  583 = 'S3 583 Row 59 Lost Return Position... Check Ixxx.x Default' | German: 'S3 583 Row 59 Lost Return Position... Check Ixxx.x German' | French: 'S3 583 Row 59 Lost Return Position... Check Ixxx.x French'
  584 = 'S3 584 Row 59 Switch Fault... Check Ixxx.x / Ixxx.x Default' | German: 'S3 584 Row 59 Switch Fault... Check Ixxx.x / Ixxx.x German' | French: 'S3 584 Row 59 Switch Fault... Check Ixxx.x / Ixxx.x French'
  585 = 'S3 585 Row 59 Spare Message Default' | German: 'S3 585 Row 59 Spare Message German' | French: 'S3 585 Row 59 Spare Message French'
  586 = 'S3 586 Row 59 Spare Message Default' | German: 'S3 586 Row 59 Spare Message German' | French: 'S3 586 Row 59 Spare Message French'
  587 = 'S3 587 Row 59 Spare Message Default' | German: 'S3 587 Row 59 Spare Message German' | French: 'S3 587 Row 59 Spare Message French'
  588 = 'S3 588 Row 59 Spare Message Default' | German: 'S3 588 Row 59 Spare Message German' | French: 'S3 588 Row 59 Spare Message French'
  589 = 'S3 589 Row 59 Spare Message Default' | German: 'S3 589 Row 59 Spare Message German' | French: 'S3 589 Row 59 Spare Message French'
  590 = 'S3 590 Row 60 Failed To Advance.. Check Qxxx.x Default' | German: 'S3 590 Row 60 Failed To Advance.. Check Qxxx.x German' | French: 'S3 590 Row 60 Failed To Advance.. Check Qxxx.x French'
  591 = 'S3 591 Row 60 Failed To Return.. Check Qxxx.x Default' | German: 'S3 591 Row 60 Failed To Return.. Check Qxxx.x German' | French: 'S3 591 Row 60 Failed To Return.. Check Qxxx.x French'
  592 = 'S3 592 Row 60 Lost Advance Position... Check Ixxx.x Default' | German: 'S3 592 Row 60 Lost Advance Position... Check Ixxx.x German' | French: 'S3 592 Row 60 Lost Advance Position... Check Ixxx.x French'
  593 = 'S3 593 Row 60 Lost Return Position... Check Ixxx.x Default' | German: 'S3 593 Row 60 Lost Return Position... Check Ixxx.x German' | French: 'S3 593 Row 60 Lost Return Position... Check Ixxx.x French'
  594 = 'S3 594 Row 60 Switch Fault... Check Ixxx.x / Ixxx.x Default' | German: 'S3 594 Row 60 Switch Fault... Check Ixxx.x / Ixxx.x German' | French: 'S3 594 Row 60 Switch Fault... Check Ixxx.x / Ixxx.x French'
  595 = 'S3 595 Row 60 Spare Message Default' | German: 'S3 595 Row 60 Spare Message German' | French: 'S3 595 Row 60 Spare Message French'
  596 = 'S3 596 Row 60 Spare Message Default' | German: 'S3 596 Row 60 Spare Message German' | French: 'S3 596 Row 60 Spare Message French'
  597 = 'S3 597 Row 60 Spare Message Default' | German: 'S3 597 Row 60 Spare Message German' | French: 'S3 597 Row 60 Spare Message French'
  598 = 'S3 598 Row 60 Spare Message Default' | German: 'S3 598 Row 60 Spare Message German' | French: 'S3 598 Row 60 Spare Message French'
  599 = 'S3 599 Row 60 Spare Message Default' | German: 'S3 599 Row 60 Spare Message German' | French: 'S3 599 Row 60 Spare Message French'
  600 = 'S3 600 Row 61 Failed To Advance.. Check Qxxx.x Default' | German: 'S3 600 Row 61 Failed To Advance.. Check Qxxx.x German' | French: 'S3 600 Row 61 Failed To Advance.. Check Qxxx.x French'
  601 = 'S3 601 Row 61 Failed To Return.. Check Qxxx.x Default' | German: 'S3 601 Row 61 Failed To Return.. Check Qxxx.x German' | French: 'S3 601 Row 61 Failed To Return.. Check Qxxx.x French'
  602 = 'S3 602 Row 61 Lost Advance Position... Check Ixxx.x Default' | German: 'S3 602 Row 61 Lost Advance Position... Check Ixxx.x German' | French: 'S3 602 Row 61 Lost Advance Position... Check Ixxx.x French'
  603 = 'S3 603 Row 61 Lost Return Position... Check Ixxx.x Default' | German: 'S3 603 Row 61 Lost Return Position... Check Ixxx.x German' | French: 'S3 603 Row 61 Lost Return Position... Check Ixxx.x French'
  604 = 'S3 604 Row 61 Switch Fault... Check Ixxx.x / Ixxx.x Default' | German: 'S3 604 Row 61 Switch Fault... Check Ixxx.x / Ixxx.x German' | French: 'S3 604 Row 61 Switch Fault... Check Ixxx.x / Ixxx.x French'
  605 = 'S3 605 Row 61 Spare Message Default' | German: 'S3 605 Row 61 Spare Message German' | French: 'S3 605 Row 61 Spare Message French'
  606 = 'S3 606 Row 61 Spare Message Default' | German: 'S3 606 Row 61 Spare Message German' | French: 'S3 606 Row 61 Spare Message French'
  607 = 'S3 607 Row 61 Spare Message Default' | German: 'S3 607 Row 61 Spare Message German' | French: 'S3 607 Row 61 Spare Message French'
  608 = 'S3 608 Row 61 Spare Message Default' | German: 'S3 608 Row 61 Spare Message German' | French: 'S3 608 Row 61 Spare Message French'
  609 = 'S3 609 Row 61 Spare Message Default' | German: 'S3 609 Row 61 Spare Message German' | French: 'S3 609 Row 61 Spare Message French'
  610 = 'S3 610 Row 62 Failed To Advance.. Check Qxxx.x Default' | German: 'S3 610 Row 62 Failed To Advance.. Check Qxxx.x German' | French: 'S3 610 Row 62 Failed To Advance.. Check Qxxx.x French'
  611 = 'S3 611 Row 62 Failed To Return.. Check Qxxx.x Default' | German: 'S3 611 Row 62 Failed To Return.. Check Qxxx.x German' | French: 'S3 611 Row 62 Failed To Return.. Check Qxxx.x French'
  612 = 'S3 612 Row 62 Lost Advance Position... Check Ixxx.x Default' | German: 'S3 612 Row 62 Lost Advance Position... Check Ixxx.x German' | French: 'S3 612 Row 62 Lost Advance Position... Check Ixxx.x French'
  613 = 'S3 613 Row 62 Lost Return Position... Check Ixxx.x Default' | German: 'S3 613 Row 62 Lost Return Position... Check Ixxx.x German' | French: 'S3 613 Row 62 Lost Return Position... Check Ixxx.x French'
  614 = 'S3 614 Row 62 Switch Fault... Check Ixxx.x / Ixxx.x Default' | German: 'S3 614 Row 62 Switch Fault... Check Ixxx.x / Ixxx.x German' | French: 'S3 614 Row 62 Switch Fault... Check Ixxx.x / Ixxx.x French'
  615 = 'S3 615 Row 62 Spare Message Default' | German: 'S3 615 Row 62 Spare Message German' | French: 'S3 615 Row 62 Spare Message French'
  616 = 'S3 616 Row 62 Spare Message Default' | German: 'S3 616 Row 62 Spare Message German' | French: 'S3 616 Row 62 Spare Message French'
  617 = 'S3 617 Row 62 Spare Message Default' | German: 'S3 617 Row 62 Spare Message German' | French: 'S3 617 Row 62 Spare Message French'
  618 = 'S3 618 Row 62 Spare Message Default' | German: 'S3 618 Row 62 Spare Message German' | French: 'S3 618 Row 62 Spare Message French'
  619 = 'S3 619 Row 62 Spare Message Default' | German: 'S3 619 Row 62 Spare Message German' | French: 'S3 619 Row 62 Spare Message French'
  620 = 'S3 620 Row 63 Failed To Advance.. Check Qxxx.x Default' | German: 'S3 620 Row 63 Failed To Advance.. Check Qxxx.x German' | French: 'S3 620 Row 63 Failed To Advance.. Check Qxxx.x French'
  621 = 'S3 621 Row 63 Failed To Return.. Check Qxxx.x Default' | German: 'S3 621 Row 63 Failed To Return.. Check Qxxx.x German' | French: 'S3 621 Row 63 Failed To Return.. Check Qxxx.x French'
  622 = 'S3 622 Row 63 Lost Advance Position... Check Ixxx.x Default' | German: 'S3 622 Row 63 Lost Advance Position... Check Ixxx.x German' | French: 'S3 622 Row 63 Lost Advance Position... Check Ixxx.x French'
  623 = 'S3 623 Row 63 Lost Return Position... Check Ixxx.x Default' | German: 'S3 623 Row 63 Lost Return Position... Check Ixxx.x German' | French: 'S3 623 Row 63 Lost Return Position... Check Ixxx.x French'
  624 = 'S3 624 Row 63 Switch Fault... Check Ixxx.x / Ixxx.x Default' | German: 'S3 624 Row 63 Switch Fault... Check Ixxx.x / Ixxx.x German' | French: 'S3 624 Row 63 Switch Fault... Check Ixxx.x / Ixxx.x French'
  625 = 'S3 625 Row 63 Spare Message Default' | German: 'S3 625 Row 63 Spare Message German' | French: 'S3 625 Row 63 Spare Message French'
  626 = 'S3 626 Row 63 Spare Message Default' | German: 'S3 626 Row 63 Spare Message German' | French: 'S3 626 Row 63 Spare Message French'
  627 = 'S3 627 Row 63 Spare Message Default' | German: 'S3 627 Row 63 Spare Message German' | French: 'S3 627 Row 63 Spare Message French'
  628 = 'S3 628 Row 63 Spare Message Default' | German: 'S3 628 Row 63 Spare Message German' | French: 'S3 628 Row 63 Spare Message French'
  629 = 'S3 629 Row 63 Spare Message Default' | German: 'S3 629 Row 63 Spare Message German' | French: 'S3 629 Row 63 Spare Message French'
  630 = 'S3 630 Row 64 Failed To Advance.. Check Qxxx.x Default' | German: 'S3 630 Row 64 Failed To Advance.. Check Qxxx.x German' | French: 'S3 630 Row 64 Failed To Advance.. Check Qxxx.x French'
  631 = 'S3 631 Row 64 Failed To Return.. Check Qxxx.x Default' | German: 'S3 631 Row 64 Failed To Return.. Check Qxxx.x German' | French: 'S3 631 Row 64 Failed To Return.. Check Qxxx.x French'
  632 = 'S3 632 Row 64 Lost Advance Position... Check Ixxx.x Default' | German: 'S3 632 Row 64 Lost Advance Position... Check Ixxx.x German' | French: 'S3 632 Row 64 Lost Advance Position... Check Ixxx.x French'
  633 = 'S3 633 Row 64 Lost Return Position... Check Ixxx.x Default' | German: 'S3 633 Row 64 Lost Return Position... Check Ixxx.x German' | French: 'S3 633 Row 64 Lost Return Position... Check Ixxx.x French'
  634 = 'S3 634 Row 64 Switch Fault... Check Ixxx.x / Ixxx.x Default' | German: 'S3 634 Row 64 Switch Fault... Check Ixxx.x / Ixxx.x German' | French: 'S3 634 Row 64 Switch Fault... Check Ixxx.x / Ixxx.x French'
  635 = 'S3 635 Row 64 Spare Message Default' | German: 'S3 635 Row 64 Spare Message German' | French: 'S3 635 Row 64 Spare Message French'
  636 = 'S3 636 Row 64 Spare Message Default' | German: 'S3 636 Row 64 Spare Message German' | French: 'S3 636 Row 64 Spare Message French'
  637 = 'S3 637 Row 64 Spare Message Default' | German: 'S3 637 Row 64 Spare Message German' | French: 'S3 637 Row 64 Spare Message French'
  638 = 'S3 638 Row 64 Spare Message Default' | German: 'S3 638 Row 64 Spare Message German' | French: 'S3 638 Row 64 Spare Message French'
  639 = 'S3 639 Row 64 Spare Message Default' | German: 'S3 639 Row 64 Spare Message German' | French: 'S3 639 Row 64 Spare Message French'
  640 = 'S3 640 Row 65 Failed To Advance.. Check Qxxx.x Default' | German: 'S3 640 Row 65 Failed To Advance.. Check Qxxx.x German' | French: 'S3 640 Row 65 Failed To Advance.. Check Qxxx.x French'
  641 = 'S3 641 Row 65 Failed To Return.. Check Qxxx.x Default' | German: 'S3 641 Row 65 Failed To Return.. Check Qxxx.x German' | French: 'S3 641 Row 65 Failed To Return.. Check Qxxx.x French'
  642 = 'S3 642 Row 65 Lost Advance Position... Check Ixxx.x Default' | German: 'S3 642 Row 65 Lost Advance Position... Check Ixxx.x German' | French: 'S3 642 Row 65 Lost Advance Position... Check Ixxx.x French'
  643 = 'S3 643 Row 65 Lost Return Position... Check Ixxx.x Default' | German: 'S3 643 Row 65 Lost Return Position... Check Ixxx.x German' | French: 'S3 643 Row 65 Lost Return Position... Check Ixxx.x French'
  644 = 'S3 644 Row 65 Switch Fault... Check Ixxx.x / Ixxx.x Default' | German: 'S3 644 Row 65 Switch Fault... Check Ixxx.x / Ixxx.x German' | French: 'S3 644 Row 65 Switch Fault... Check Ixxx.x / Ixxx.x French'
  645 = 'S3 645 Row 65 Spare Message Default' | German: 'S3 645 Row 65 Spare Message German' | French: 'S3 645 Row 65 Spare Message French'
  646 = 'S3 646 Row 65 Spare Message Default' | German: 'S3 646 Row 65 Spare Message German' | French: 'S3 646 Row 65 Spare Message French'
  647 = 'S3 647 Row 65 Spare Message Default' | German: 'S3 647 Row 65 Spare Message German' | French: 'S3 647 Row 65 Spare Message French'
  648 = 'S3 648 Row 65 Spare Message Default' | German: 'S3 648 Row 65 Spare Message German' | French: 'S3 648 Row 65 Spare Message French'
  649 = 'S3 649 Row 65 Spare Message Default' | German: 'S3 649 Row 65 Spare Message German' | French: 'S3 649 Row 65 Spare Message French'
  650 = 'S3 650 Row 66 Failed To Advance.. Check Qxxx.x Default' | German: 'S3 650 Row 66 Failed To Advance.. Check Qxxx.x German' | French: 'S3 650 Row 66 Failed To Advance.. Check Qxxx.x French'
  651 = 'S3 651 Row 66 Failed To Return.. Check Qxxx.x Default' | German: 'S3 651 Row 66 Failed To Return.. Check Qxxx.x German' | French: 'S3 651 Row 66 Failed To Return.. Check Qxxx.x French'
  652 = 'S3 652 Row 66 Lost Advance Position... Check Ixxx.x Default' | German: 'S3 652 Row 66 Lost Advance Position... Check Ixxx.x German' | French: 'S3 652 Row 66 Lost Advance Position... Check Ixxx.x French'
  653 = 'S3 653 Row 66 Lost Return Position... Check Ixxx.x Default' | German: 'S3 653 Row 66 Lost Return Position... Check Ixxx.x German' | French: 'S3 653 Row 66 Lost Return Position... Check Ixxx.x French'
  654 = 'S3 654 Row 66 Switch Fault... Check Ixxx.x / Ixxx.x Default' | German: 'S3 654 Row 66 Switch Fault... Check Ixxx.x / Ixxx.x German' | French: 'S3 654 Row 66 Switch Fault... Check Ixxx.x / Ixxx.x French'
  655 = 'S3 655 Row 66 Spare Message Default' | German: 'S3 655 Row 66 Spare Message German' | French: 'S3 655 Row 66 Spare Message French'
  656 = 'S3 656 Row 66 Spare Message Default' | German: 'S3 656 Row 66 Spare Message German' | French: 'S3 656 Row 66 Spare Message French'
  657 = 'S3 657 Row 66 Spare Message Default' | German: 'S3 657 Row 66 Spare Message German' | French: 'S3 657 Row 66 Spare Message French'
  658 = 'S3 658 Row 66 Spare Message Default' | German: 'S3 658 Row 66 Spare Message German' | French: 'S3 658 Row 66 Spare Message French'
  659 = 'S3 659 Row 66 Spare Message Default' | German: 'S3 659 Row 66 Spare Message German' | French: 'S3 659 Row 66 Spare Message French'
  660 = 'S3 660 Row 67 Failed To Advance.. Check Qxxx.x Default' | German: 'S3 660 Row 67 Failed To Advance.. Check Qxxx.x German' | French: 'S3 660 Row 67 Failed To Advance.. Check Qxxx.x French'
  661 = 'S3 661 Row 67 Failed To Return.. Check Qxxx.x Default' | German: 'S3 661 Row 67 Failed To Return.. Check Qxxx.x German' | French: 'S3 661 Row 67 Failed To Return.. Check Qxxx.x French'
  662 = 'S3 662 Row 67 Lost Advance Position... Check Ixxx.x Default' | German: 'S3 662 Row 67 Lost Advance Position... Check Ixxx.x German' | French: 'S3 662 Row 67 Lost Advance Position... Check Ixxx.x French'
  663 = 'S3 663 Row 67 Lost Return Position... Check Ixxx.x Default' | German: 'S3 663 Row 67 Lost Return Position... Check Ixxx.x German' | French: 'S3 663 Row 67 Lost Return Position... Check Ixxx.x French'
  664 = 'S3 664 Row 67 Switch Fault... Check Ixxx.x / Ixxx.x Default' | German: 'S3 664 Row 67 Switch Fault... Check Ixxx.x / Ixxx.x German' | French: 'S3 664 Row 67 Switch Fault... Check Ixxx.x / Ixxx.x French'
  665 = 'S3 665 Row 67 Spare Message Default' | German: 'S3 665 Row 67 Spare Message German' | French: 'S3 665 Row 67 Spare Message French'
  666 = 'S3 666 Row 67 Spare Message Default' | German: 'S3 666 Row 67 Spare Message German' | French: 'S3 666 Row 67 Spare Message French'
  667 = 'S3 667 Row 67 Spare Message Default' | German: 'S3 667 Row 67 Spare Message German' | French: 'S3 667 Row 67 Spare Message French'
  668 = 'S3 668 Row 67 Spare Message Default' | German: 'S3 668 Row 67 Spare Message German' | French: 'S3 668 Row 67 Spare Message French'
  669 = 'S3 669 Row 67 Spare Message Default' | German: 'S3 669 Row 67 Spare Message German' | French: 'S3 669 Row 67 Spare Message French'
  670 = 'S3 670 Row 68 Failed To Advance.. Check Qxxx.x Default' | German: 'S3 670 Row 68 Failed To Advance.. Check Qxxx.x German' | French: 'S3 670 Row 68 Failed To Advance.. Check Qxxx.x French'
  671 = 'S3 671 Row 68 Failed To Return.. Check Qxxx.x Default' | German: 'S3 671 Row 68 Failed To Return.. Check Qxxx.x German' | French: 'S3 671 Row 68 Failed To Return.. Check Qxxx.x French'
  672 = 'S3 672 Row 68 Lost Advance Position... Check Ixxx.x Default' | German: 'S3 672 Row 68 Lost Advance Position... Check Ixxx.x German' | French: 'S3 672 Row 68 Lost Advance Position... Check Ixxx.x French'
  673 = 'S3 673 Row 68 Lost Return Position... Check Ixxx.x Default' | German: 'S3 673 Row 68 Lost Return Position... Check Ixxx.x German' | French: 'S3 673 Row 68 Lost Return Position... Check Ixxx.x French'
  674 = 'S3 674 Row 68 Switch Fault... Check Ixxx.x / Ixxx.x Default' | German: 'S3 674 Row 68 Switch Fault... Check Ixxx.x / Ixxx.x German' | French: 'S3 674 Row 68 Switch Fault... Check Ixxx.x / Ixxx.x French'
  675 = 'S3 675 Row 68 Spare Message Default' | German: 'S3 675 Row 68 Spare Message German' | French: 'S3 675 Row 68 Spare Message French'
  676 = 'S3 676 Row 68 Spare Message Default' | German: 'S3 676 Row 68 Spare Message German' | French: 'S3 676 Row 68 Spare Message French'
  677 = 'S3 677 Row 68 Spare Message Default' | German: 'S3 677 Row 68 Spare Message German' | French: 'S3 677 Row 68 Spare Message French'
  678 = 'S3 678 Row 68 Spare Message Default' | German: 'S3 678 Row 68 Spare Message German' | French: 'S3 678 Row 68 Spare Message French'
  679 = 'S3 679 Row 68 Spare Message Default' | German: 'S3 679 Row 68 Spare Message German' | French: 'S3 679 Row 68 Spare Message French'
  680 = 'S3 680 Row 69 Failed To Advance.. Check Qxxx.x Default' | German: 'S3 680 Row 69 Failed To Advance.. Check Qxxx.x German' | French: 'S3 680 Row 69 Failed To Advance.. Check Qxxx.x French'
  681 = 'S3 681 Row 69 Failed To Return.. Check Qxxx.x Default' | German: 'S3 681 Row 69 Failed To Return.. Check Qxxx.x German' | French: 'S3 681 Row 69 Failed To Return.. Check Qxxx.x French'
  682 = 'S3 682 Row 69 Lost Advance Position... Check Ixxx.x Default' | German: 'S3 682 Row 69 Lost Advance Position... Check Ixxx.x German' | French: 'S3 682 Row 69 Lost Advance Position... Check Ixxx.x French'
  683 = 'S3 683 Row 69 Lost Return Position... Check Ixxx.x Default' | German: 'S3 683 Row 69 Lost Return Position... Check Ixxx.x German' | French: 'S3 683 Row 69 Lost Return Position... Check Ixxx.x French'
  684 = 'S3 684 Row 69 Switch Fault... Check Ixxx.x / Ixxx.x Default' | German: 'S3 684 Row 69 Switch Fault... Check Ixxx.x / Ixxx.x German' | French: 'S3 684 Row 69 Switch Fault... Check Ixxx.x / Ixxx.x French'
  685 = 'S3 685 Row 69 Spare Message Default' | German: 'S3 685 Row 69 Spare Message German' | French: 'S3 685 Row 69 Spare Message French'
  686 = 'S3 686 Row 69 Spare Message Default' | German: 'S3 686 Row 69 Spare Message German' | French: 'S3 686 Row 69 Spare Message French'
  687 = 'S3 687 Row 69 Spare Message Default' | German: 'S3 687 Row 69 Spare Message German' | French: 'S3 687 Row 69 Spare Message French'
  688 = 'S3 688 Row 69 Spare Message Default' | German: 'S3 688 Row 69 Spare Message German' | French: 'S3 688 Row 69 Spare Message French'
  689 = 'S3 689 Row 69 Spare Message Default' | German: 'S3 689 Row 69 Spare Message German' | French: 'S3 689 Row 69 Spare Message French'
  690 = 'S3 690 Row 70 Failed To Advance.. Check Qxxx.x Default' | German: 'S3 690 Row 70 Failed To Advance.. Check Qxxx.x German' | French: 'S3 690 Row 70 Failed To Advance.. Check Qxxx.x French'
  691 = 'S3 691 Row 70 Failed To Return.. Check Qxxx.x Default' | German: 'S3 691 Row 70 Failed To Return.. Check Qxxx.x German' | French: 'S3 691 Row 70 Failed To Return.. Check Qxxx.x French'
  692 = 'S3 692 Row 70 Lost Advance Position... Check Ixxx.x Default' | German: 'S3 692 Row 70 Lost Advance Position... Check Ixxx.x German' | French: 'S3 692 Row 70 Lost Advance Position... Check Ixxx.x French'
  693 = 'S3 693 Row 70 Lost Return Position... Check Ixxx.x Default' | German: 'S3 693 Row 70 Lost Return Position... Check Ixxx.x German' | French: 'S3 693 Row 70 Lost Return Position... Check Ixxx.x French'
  694 = 'S3 694 Row 70 Switch Fault... Check Ixxx.x / Ixxx.x Default' | German: 'S3 694 Row 70 Switch Fault... Check Ixxx.x / Ixxx.x German' | French: 'S3 694 Row 70 Switch Fault... Check Ixxx.x / Ixxx.x French'
  695 = 'S3 695 Row 70 Spare Message Default' | German: 'S3 695 Row 70 Spare Message German' | French: 'S3 695 Row 70 Spare Message French'
  696 = 'S3 696 Row 70 Spare Message Default' | German: 'S3 696 Row 70 Spare Message German' | French: 'S3 696 Row 70 Spare Message French'
  697 = 'S3 697 Row 70 Spare Message Default' | German: 'S3 697 Row 70 Spare Message German' | French: 'S3 697 Row 70 Spare Message French'
  698 = 'S3 698 Row 70 Spare Message Default' | German: 'S3 698 Row 70 Spare Message German' | French: 'S3 698 Row 70 Spare Message French'
  699 = 'S3 699 Row 70 Spare Message Default' | German: 'S3 699 Row 70 Spare Message German' | French: 'S3 699 Row 70 Spare Message French'
  700 = 'S3 700 Row 71 Failed To Advance.. Check Qxxx.x Default' | German: 'S3 700 Row 71 Failed To Advance.. Check Qxxx.x German' | French: 'S3 700 Row 71 Failed To Advance.. Check Qxxx.x French'
  701 = 'S3 701 Row 71 Failed To Return.. Check Qxxx.x Default' | German: 'S3 701 Row 71 Failed To Return.. Check Qxxx.x German' | French: 'S3 701 Row 71 Failed To Return.. Check Qxxx.x French'
  702 = 'S3 702 Row 71 Lost Advance Position... Check Ixxx.x Default' | German: 'S3 702 Row 71 Lost Advance Position... Check Ixxx.x German' | French: 'S3 702 Row 71 Lost Advance Position... Check Ixxx.x French'
  703 = 'S3 703 Row 71 Lost Return Position... Check Ixxx.x Default' | German: 'S3 703 Row 71 Lost Return Position... Check Ixxx.x German' | French: 'S3 703 Row 71 Lost Return Position... Check Ixxx.x French'
  704 = 'S3 704 Row 71 Switch Fault... Check Ixxx.x / Ixxx.x Default' | German: 'S3 704 Row 71 Switch Fault... Check Ixxx.x / Ixxx.x German' | French: 'S3 704 Row 71 Switch Fault... Check Ixxx.x / Ixxx.x French'
  705 = 'S3 705 Row 71 Spare Message Default' | German: 'S3 705 Row 71 Spare Message German' | French: 'S3 705 Row 71 Spare Message French'
  706 = 'S3 706 Row 71 Spare Message Default' | German: 'S3 706 Row 71 Spare Message German' | French: 'S3 706 Row 71 Spare Message French'
  707 = 'S3 707 Row 71 Spare Message Default' | German: 'S3 707 Row 71 Spare Message German' | French: 'S3 707 Row 71 Spare Message French'
  708 = 'S3 708 Row 71 Spare Message Default' | German: 'S3 708 Row 71 Spare Message German' | French: 'S3 708 Row 71 Spare Message French'
  709 = 'S3 709 Row 71 Spare Message Default' | German: 'S3 709 Row 71 Spare Message German' | French: 'S3 709 Row 71 Spare Message French'
  710 = 'S3 710 Row 72 Failed To Advance.. Check Qxxx.x Default' | German: 'S3 710 Row 72 Failed To Advance.. Check Qxxx.x German' | French: 'S3 710 Row 72 Failed To Advance.. Check Qxxx.x French'
  711 = 'S3 711 Row 72 Failed To Return.. Check Qxxx.x Default' | German: 'S3 711 Row 72 Failed To Return.. Check Qxxx.x German' | French: 'S3 711 Row 72 Failed To Return.. Check Qxxx.x French'
  712 = 'S3 712 Row 72 Lost Advance Position... Check Ixxx.x Default' | German: 'S3 712 Row 72 Lost Advance Position... Check Ixxx.x German' | French: 'S3 712 Row 72 Lost Advance Position... Check Ixxx.x French'
  713 = 'S3 713 Row 72 Lost Return Position... Check Ixxx.x Default' | German: 'S3 713 Row 72 Lost Return Position... Check Ixxx.x German' | French: 'S3 713 Row 72 Lost Return Position... Check Ixxx.x French'
  714 = 'S3 714 Row 72 Switch Fault... Check Ixxx.x / Ixxx.x Default' | German: 'S3 714 Row 72 Switch Fault... Check Ixxx.x / Ixxx.x German' | French: 'S3 714 Row 72 Switch Fault... Check Ixxx.x / Ixxx.x French'
  715 = 'S3 715 Row 72 Spare Message Default' | German: 'S3 715 Row 72 Spare Message German' | French: 'S3 715 Row 72 Spare Message French'
  716 = 'S3 716 Row 72 Spare Message Default' | German: 'S3 716 Row 72 Spare Message German' | French: 'S3 716 Row 72 Spare Message French'
  717 = 'S3 717 Row 72 Spare Message Default' | German: 'S3 717 Row 72 Spare Message German' | French: 'S3 717 Row 72 Spare Message French'
  718 = 'S3 718 Row 72 Spare Message Default' | German: 'S3 718 Row 72 Spare Message German' | French: 'S3 718 Row 72 Spare Message French'
  719 = 'S3 719 Row 72 Spare Message Default' | German: 'S3 719 Row 72 Spare Message German' | French: 'S3 719 Row 72 Spare Message French'
  720 = 'S3 720 Row 73 Failed To Advance.. Check Qxxx.x Default' | German: 'S3 720 Row 73 Failed To Advance.. Check Qxxx.x German' | French: 'S3 720 Row 73 Failed To Advance.. Check Qxxx.x French'
  721 = 'S3 721 Row 73 Failed To Return.. Check Qxxx.x Default' | German: 'S3 721 Row 73 Failed To Return.. Check Qxxx.x German' | French: 'S3 721 Row 73 Failed To Return.. Check Qxxx.x French'
  722 = 'S3 722 Row 73 Lost Advance Position... Check Ixxx.x Default' | German: 'S3 722 Row 73 Lost Advance Position... Check Ixxx.x German' | French: 'S3 722 Row 73 Lost Advance Position... Check Ixxx.x French'
  723 = 'S3 723 Row 73 Lost Return Position... Check Ixxx.x Default' | German: 'S3 723 Row 73 Lost Return Position... Check Ixxx.x German' | French: 'S3 723 Row 73 Lost Return Position... Check Ixxx.x French'
  724 = 'S3 724 Row 73 Switch Fault... Check Ixxx.x / Ixxx.x Default' | German: 'S3 724 Row 73 Switch Fault... Check Ixxx.x / Ixxx.x German' | French: 'S3 724 Row 73 Switch Fault... Check Ixxx.x / Ixxx.x French'
  725 = 'S3 725 Row 73 Spare Message Default' | German: 'S3 725 Row 73 Spare Message German' | French: 'S3 725 Row 73 Spare Message French'
  726 = 'S3 726 Row 73 Spare Message Default' | German: 'S3 726 Row 73 Spare Message German' | French: 'S3 726 Row 73 Spare Message French'
  727 = 'S3 727 Row 73 Spare Message Default' | German: 'S3 727 Row 73 Spare Message German' | French: 'S3 727 Row 73 Spare Message French'
  728 = 'S3 728 Row 73 Spare Message Default' | German: 'S3 728 Row 73 Spare Message German' | French: 'S3 728 Row 73 Spare Message French'
  729 = 'S3 729 Row 73 Spare Message Default' | German: 'S3 729 Row 73 Spare Message German' | French: 'S3 729 Row 73 Spare Message French'
  730 = 'S3 730 Row 74 Failed To Advance.. Check Qxxx.x Default' | German: 'S3 730 Row 74 Failed To Advance.. Check Qxxx.x German' | French: 'S3 730 Row 74 Failed To Advance.. Check Qxxx.x French'
  731 = 'S3 731 Row 74 Failed To Return.. Check Qxxx.x Default' | German: 'S3 731 Row 74 Failed To Return.. Check Qxxx.x German' | French: 'S3 731 Row 74 Failed To Return.. Check Qxxx.x French'
  732 = 'S3 732 Row 74 Lost Advance Position... Check Ixxx.x Default' | German: 'S3 732 Row 74 Lost Advance Position... Check Ixxx.x German' | French: 'S3 732 Row 74 Lost Advance Position... Check Ixxx.x French'
  733 = 'S3 733 Row 74 Lost Return Position... Check Ixxx.x Default' | German: 'S3 733 Row 74 Lost Return Position... Check Ixxx.x German' | French: 'S3 733 Row 74 Lost Return Position... Check Ixxx.x French'
  734 = 'S3 734 Row 74 Switch Fault... Check Ixxx.x / Ixxx.x Default' | German: 'S3 734 Row 74 Switch Fault... Check Ixxx.x / Ixxx.x German' | French: 'S3 734 Row 74 Switch Fault... Check Ixxx.x / Ixxx.x French'
  735 = 'S3 735 Row 74 Spare Message Default' | German: 'S3 735 Row 74 Spare Message German' | French: 'S3 735 Row 74 Spare Message French'
  736 = 'S3 736 Row 74 Spare Message Default' | German: 'S3 736 Row 74 Spare Message German' | French: 'S3 736 Row 74 Spare Message French'
  737 = 'S3 737 Row 74 Spare Message Default' | German: 'S3 737 Row 74 Spare Message German' | French: 'S3 737 Row 74 Spare Message French'
  738 = 'S3 738 Row 74 Spare Message Default' | German: 'S3 738 Row 74 Spare Message German' | French: 'S3 738 Row 74 Spare Message French'
  739 = 'S3 739 Row 74 Spare Message Default' | German: 'S3 739 Row 74 Spare Message German' | French: 'S3 739 Row 74 Spare Message French'
  740 = 'S3 740 Row 75 Failed To Advance.. Check Qxxx.x Default' | German: 'S3 740 Row 75 Failed To Advance.. Check Qxxx.x German' | French: 'S3 740 Row 75 Failed To Advance.. Check Qxxx.x French'
  741 = 'S3 741 Row 75 Failed To Return.. Check Qxxx.x Default' | German: 'S3 741 Row 75 Failed To Return.. Check Qxxx.x German' | French: 'S3 741 Row 75 Failed To Return.. Check Qxxx.x French'
  742 = 'S3 742 Row 75 Lost Advance Position... Check Ixxx.x Default' | German: 'S3 742 Row 75 Lost Advance Position... Check Ixxx.x German' | French: 'S3 742 Row 75 Lost Advance Position... Check Ixxx.x French'
  743 = 'S3 743 Row 75 Lost Return Position... Check Ixxx.x Default' | German: 'S3 743 Row 75 Lost Return Position... Check Ixxx.x German' | French: 'S3 743 Row 75 Lost Return Position... Check Ixxx.x French'
  744 = 'S3 744 Row 75 Switch Fault... Check Ixxx.x / Ixxx.x Default' | German: 'S3 744 Row 75 Switch Fault... Check Ixxx.x / Ixxx.x German' | French: 'S3 744 Row 75 Switch Fault... Check Ixxx.x / Ixxx.x French'
  745 = 'S3 745 Row 75 Spare Message Default' | German: 'S3 745 Row 75 Spare Message German' | French: 'S3 745 Row 75 Spare Message French'
  746 = 'S3 746 Row 75 Spare Message Default' | German: 'S3 746 Row 75 Spare Message German' | French: 'S3 746 Row 75 Spare Message French'
  747 = 'S3 747 Row 75 Spare Message Default' | German: 'S3 747 Row 75 Spare Message German' | French: 'S3 747 Row 75 Spare Message French'
  748 = 'S3 748 Row 75 Spare Message Default' | German: 'S3 748 Row 75 Spare Message German' | French: 'S3 748 Row 75 Spare Message French'
  749 = 'S3 749 Row 75 Spare Message Default' | German: 'S3 749 Row 75 Spare Message German' | French: 'S3 749 Row 75 Spare Message French'
  750 = 'S3 750 Row 76 Failed To Advance.. Check Qxxx.x Default' | German: 'S3 750 Row 76 Failed To Advance.. Check Qxxx.x German' | French: 'S3 750 Row 76 Failed To Advance.. Check Qxxx.x French'
  751 = 'S3 751 Row 76 Failed To Return.. Check Qxxx.x Default' | German: 'S3 751 Row 76 Failed To Return.. Check Qxxx.x German' | French: 'S3 751 Row 76 Failed To Return.. Check Qxxx.x French'
  752 = 'S3 752 Row 76 Lost Advance Position... Check Ixxx.x Default' | German: 'S3 752 Row 76 Lost Advance Position... Check Ixxx.x German' | French: 'S3 752 Row 76 Lost Advance Position... Check Ixxx.x French'
  753 = 'S3 753 Row 76 Lost Return Position... Check Ixxx.x Default' | German: 'S3 753 Row 76 Lost Return Position... Check Ixxx.x German' | French: 'S3 753 Row 76 Lost Return Position... Check Ixxx.x French'
  754 = 'S3 754 Row 76 Switch Fault... Check Ixxx.x / Ixxx.x Default' | German: 'S3 754 Row 76 Switch Fault... Check Ixxx.x / Ixxx.x German' | French: 'S3 754 Row 76 Switch Fault... Check Ixxx.x / Ixxx.x French'
  755 = 'S3 755 Row 76 Spare Message Default' | German: 'S3 755 Row 76 Spare Message German' | French: 'S3 755 Row 76 Spare Message French'
  756 = 'S3 756 Row 76 Spare Message Default' | German: 'S3 756 Row 76 Spare Message German' | French: 'S3 756 Row 76 Spare Message French'
  757 = 'S3 757 Row 76 Spare Message Default' | German: 'S3 757 Row 76 Spare Message German' | French: 'S3 757 Row 76 Spare Message French'
  758 = 'S3 758 Row 76 Spare Message Default' | German: 'S3 758 Row 76 Spare Message German' | French: 'S3 758 Row 76 Spare Message French'
  759 = 'S3 759 Row 76 Spare Message Default' | German: 'S3 759 Row 76 Spare Message German' | French: 'S3 759 Row 76 Spare Message French'
  760 = 'S3 760 Row 77 Failed To Advance.. Check Qxxx.x Default' | German: 'S3 760 Row 77 Failed To Advance.. Check Qxxx.x German' | French: 'S3 760 Row 77 Failed To Advance.. Check Qxxx.x French'
  761 = 'S3 761 Row 77 Failed To Return.. Check Qxxx.x Default' | German: 'S3 761 Row 77 Failed To Return.. Check Qxxx.x German' | French: 'S3 761 Row 77 Failed To Return.. Check Qxxx.x French'
  762 = 'S3 762 Row 77 Lost Advance Position... Check Ixxx.x Default' | German: 'S3 762 Row 77 Lost Advance Position... Check Ixxx.x German' | French: 'S3 762 Row 77 Lost Advance Position... Check Ixxx.x French'
  763 = 'S3 763 Row 77 Lost Return Position... Check Ixxx.x Default' | German: 'S3 763 Row 77 Lost Return Position... Check Ixxx.x German' | French: 'S3 763 Row 77 Lost Return Position... Check Ixxx.x French'
  764 = 'S3 764 Row 77 Switch Fault... Check Ixxx.x / Ixxx.x Default' | German: 'S3 764 Row 77 Switch Fault... Check Ixxx.x / Ixxx.x German' | French: 'S3 764 Row 77 Switch Fault... Check Ixxx.x / Ixxx.x French'
  765 = 'S3 765 Row 77 Spare Message Default' | German: 'S3 765 Row 77 Spare Message German' | French: 'S3 765 Row 77 Spare Message French'
  766 = 'S3 766 Row 77 Spare Message Default' | German: 'S3 766 Row 77 Spare Message German' | French: 'S3 766 Row 77 Spare Message French'
  767 = 'S3 767 Row 77 Spare Message Default' | German: 'S3 767 Row 77 Spare Message German' | French: 'S3 767 Row 77 Spare Message French'
  768 = 'S3 768 Row 77 Spare Message Default' | German: 'S3 768 Row 77 Spare Message German' | French: 'S3 768 Row 77 Spare Message French'
  769 = 'S3 769 Row 77 Spare Message Default' | German: 'S3 769 Row 77 Spare Message German' | French: 'S3 769 Row 77 Spare Message French'
  770 = 'S3 770 Row 78 Failed To Advance.. Check Qxxx.x Default' | German: 'S3 770 Row 78 Failed To Advance.. Check Qxxx.x German' | French: 'S3 770 Row 78 Failed To Advance.. Check Qxxx.x French'
  771 = 'S3 771 Row 78 Failed To Return.. Check Qxxx.x Default' | German: 'S3 771 Row 78 Failed To Return.. Check Qxxx.x German' | French: 'S3 771 Row 78 Failed To Return.. Check Qxxx.x French'
  772 = 'S3 772 Row 78 Lost Advance Position... Check Ixxx.x Default' | German: 'S3 772 Row 78 Lost Advance Position... Check Ixxx.x German' | French: 'S3 772 Row 78 Lost Advance Position... Check Ixxx.x French'
  773 = 'S3 773 Row 78 Lost Return Position... Check Ixxx.x Default' | German: 'S3 773 Row 78 Lost Return Position... Check Ixxx.x German' | French: 'S3 773 Row 78 Lost Return Position... Check Ixxx.x French'
  774 = 'S3 774 Row 78 Switch Fault... Check Ixxx.x / Ixxx.x Default' | German: 'S3 774 Row 78 Switch Fault... Check Ixxx.x / Ixxx.x German' | French: 'S3 774 Row 78 Switch Fault... Check Ixxx.x / Ixxx.x French'
  775 = 'S3 775 Row 78 Spare Message Default' | German: 'S3 775 Row 78 Spare Message German' | French: 'S3 775 Row 78 Spare Message French'
  776 = 'S3 776 Row 78 Spare Message Default' | German: 'S3 776 Row 78 Spare Message German' | French: 'S3 776 Row 78 Spare Message French'
  777 = 'S3 777 Row 78 Spare Message Default' | German: 'S3 777 Row 78 Spare Message German' | French: 'S3 777 Row 78 Spare Message French'
  778 = 'S3 778 Row 78 Spare Message Default' | German: 'S3 778 Row 78 Spare Message German' | French: 'S3 778 Row 78 Spare Message French'
  779 = 'S3 779 Row 78 Spare Message Default' | German: 'S3 779 Row 78 Spare Message German' | French: 'S3 779 Row 78 Spare Message French'
  780 = 'S3 780 Row 79 Failed To Advance.. Check Qxxx.x Default' | German: 'S3 780 Row 79 Failed To Advance.. Check Qxxx.x German' | French: 'S3 780 Row 79 Failed To Advance.. Check Qxxx.x French'
  781 = 'S3 781 Row 79 Failed To Return.. Check Qxxx.x Default' | German: 'S3 781 Row 79 Failed To Return.. Check Qxxx.x German' | French: 'S3 781 Row 79 Failed To Return.. Check Qxxx.x French'
  782 = 'S3 782 Row 79 Lost Advance Position... Check Ixxx.x Default' | German: 'S3 782 Row 79 Lost Advance Position... Check Ixxx.x German' | French: 'S3 782 Row 79 Lost Advance Position... Check Ixxx.x French'
  783 = 'S3 783 Row 79 Lost Return Position... Check Ixxx.x Default' | German: 'S3 783 Row 79 Lost Return Position... Check Ixxx.x German' | French: 'S3 783 Row 79 Lost Return Position... Check Ixxx.x French'
  784 = 'S3 784 Row 79 Switch Fault... Check Ixxx.x / Ixxx.x Default' | German: 'S3 784 Row 79 Switch Fault... Check Ixxx.x / Ixxx.x German' | French: 'S3 784 Row 79 Switch Fault... Check Ixxx.x / Ixxx.x French'
  785 = 'S3 785 Row 79 Spare Message Default' | German: 'S3 785 Row 79 Spare Message German' | French: 'S3 785 Row 79 Spare Message French'
  786 = 'S3 786 Row 79 Spare Message Default' | German: 'S3 786 Row 79 Spare Message German' | French: 'S3 786 Row 79 Spare Message French'
  787 = 'S3 787 Row 79 Spare Message Default' | German: 'S3 787 Row 79 Spare Message German' | French: 'S3 787 Row 79 Spare Message French'
  788 = 'S3 788 Row 79 Spare Message Default' | German: 'S3 788 Row 79 Spare Message German' | French: 'S3 788 Row 79 Spare Message French'
  789 = 'S3 789 Row 79 Spare Message Default' | German: 'S3 789 Row 79 Spare Message German' | French: 'S3 789 Row 79 Spare Message French'
  790 = 'S3 790 Row 80 Failed To Advance.. Check Qxxx.x Default' | German: 'S3 790 Row 80 Failed To Advance.. Check Qxxx.x German' | French: 'S3 790 Row 80 Failed To Advance.. Check Qxxx.x French'
  791 = 'S3 791 Row 80 Failed To Return.. Check Qxxx.x Default' | German: 'S3 791 Row 80 Failed To Return.. Check Qxxx.x German' | French: 'S3 791 Row 80 Failed To Return.. Check Qxxx.x French'
  792 = 'S3 792 Row 80 Lost Advance Position... Check Ixxx.x Default' | German: 'S3 792 Row 80 Lost Advance Position... Check Ixxx.x German' | French: 'S3 792 Row 80 Lost Advance Position... Check Ixxx.x French'
  793 = 'S3 793 Row 80 Lost Return Position... Check Ixxx.x Default' | German: 'S3 793 Row 80 Lost Return Position... Check Ixxx.x German' | French: 'S3 793 Row 80 Lost Return Position... Check Ixxx.x French'
  794 = 'S3 794 Row 80 Switch Fault... Check Ixxx.x / Ixxx.x Default' | German: 'S3 794 Row 80 Switch Fault... Check Ixxx.x / Ixxx.x German' | French: 'S3 794 Row 80 Switch Fault... Check Ixxx.x / Ixxx.x French'
  795 = 'S3 795 Row 80 Spare Message Default' | German: 'S3 795 Row 80 Spare Message German' | French: 'S3 795 Row 80 Spare Message French'
  796 = 'S3 796 Row 80 Spare Message Default' | German: 'S3 796 Row 80 Spare Message German' | French: 'S3 796 Row 80 Spare Message French'
  797 = 'S3 797 Row 80 Spare Message Default' | German: 'S3 797 Row 80 Spare Message German' | French: 'S3 797 Row 80 Spare Message French'
  798 = 'S3 798 Row 80 Spare Message Default' | German: 'S3 798 Row 80 Spare Message German' | French: 'S3 798 Row 80 Spare Message French'
  799 = 'S3 799 Row 80 Spare Message Default' | German: 'S3 799 Row 80 Spare Message German' | French: 'S3 799 Row 80 Spare Message French'
  800 = 'S3 800 Row 81 Failed To Advance.. Check Qxxx.x Default' | German: 'S3 800 Row 81 Failed To Advance.. Check Qxxx.x German' | French: 'S3 800 Row 81 Failed To Advance.. Check Qxxx.x French'
  801 = 'S3 801 Row 81 Failed To Return.. Check Qxxx.x Default' | German: 'S3 801 Row 81 Failed To Return.. Check Qxxx.x German' | French: 'S3 801 Row 81 Failed To Return.. Check Qxxx.x French'
  802 = 'S3 802 Row 81 Lost Advance Position... Check Ixxx.x Default' | German: 'S3 802 Row 81 Lost Advance Position... Check Ixxx.x German' | French: 'S3 802 Row 81 Lost Advance Position... Check Ixxx.x French'
  803 = 'S3 803 Row 81 Lost Return Position... Check Ixxx.x Default' | German: 'S3 803 Row 81 Lost Return Position... Check Ixxx.x German' | French: 'S3 803 Row 81 Lost Return Position... Check Ixxx.x French'
  804 = 'S3 804 Row 81 Switch Fault... Check Ixxx.x / Ixxx.x Default' | German: 'S3 804 Row 81 Switch Fault... Check Ixxx.x / Ixxx.x German' | French: 'S3 804 Row 81 Switch Fault... Check Ixxx.x / Ixxx.x French'
  805 = 'S3 805 Row 81 Spare Message Default' | German: 'S3 805 Row 81 Spare Message German' | French: 'S3 805 Row 81 Spare Message French'
  806 = 'S3 806 Row 81 Spare Message Default' | German: 'S3 806 Row 81 Spare Message German' | French: 'S3 806 Row 81 Spare Message French'
  807 = 'S3 807 Row 81 Spare Message Default' | German: 'S3 807 Row 81 Spare Message German' | French: 'S3 807 Row 81 Spare Message French'
  808 = 'S3 808 Row 81 Spare Message Default' | German: 'S3 808 Row 81 Spare Message German' | French: 'S3 808 Row 81 Spare Message French'
  809 = 'S3 809 Row 81 Spare Message Default' | German: 'S3 809 Row 81 Spare Message German' | French: 'S3 809 Row 81 Spare Message French'
  810 = 'S3 810 Row 82 Failed To Advance.. Check Qxxx.x Default' | German: 'S3 810 Row 82 Failed To Advance.. Check Qxxx.x German' | French: 'S3 810 Row 82 Failed To Advance.. Check Qxxx.x French'
  811 = 'S3 811 Row 82 Failed To Return.. Check Qxxx.x Default' | German: 'S3 811 Row 82 Failed To Return.. Check Qxxx.x German' | French: 'S3 811 Row 82 Failed To Return.. Check Qxxx.x French'
  812 = 'S3 812 Row 82 Lost Advance Position... Check Ixxx.x Default' | German: 'S3 812 Row 82 Lost Advance Position... Check Ixxx.x German' | French: 'S3 812 Row 82 Lost Advance Position... Check Ixxx.x French'
  813 = 'S3 813 Row 82 Lost Return Position... Check Ixxx.x Default' | German: 'S3 813 Row 82 Lost Return Position... Check Ixxx.x German' | French: 'S3 813 Row 82 Lost Return Position... Check Ixxx.x French'
  814 = 'S3 814 Row 82 Switch Fault... Check Ixxx.x / Ixxx.x Default' | German: 'S3 814 Row 82 Switch Fault... Check Ixxx.x / Ixxx.x German' | French: 'S3 814 Row 82 Switch Fault... Check Ixxx.x / Ixxx.x French'
  815 = 'S3 815 Row 82 Spare Message Default' | German: 'S3 815 Row 82 Spare Message German' | French: 'S3 815 Row 82 Spare Message French'
  816 = 'S3 816 Row 82 Spare Message Default' | German: 'S3 816 Row 82 Spare Message German' | French: 'S3 816 Row 82 Spare Message French'
  817 = 'S3 817 Row 82 Spare Message Default' | German: 'S3 817 Row 82 Spare Message German' | French: 'S3 817 Row 82 Spare Message French'
  818 = 'S3 818 Row 82 Spare Message Default' | German: 'S3 818 Row 82 Spare Message German' | French: 'S3 818 Row 82 Spare Message French'
  819 = 'S3 819 Row 82 Spare Message Default' | German: 'S3 819 Row 82 Spare Message German' | French: 'S3 819 Row 82 Spare Message French'
  820 = 'S3 820 Row 83 Failed To Advance.. Check Qxxx.x Default' | German: 'S3 820 Row 83 Failed To Advance.. Check Qxxx.x German' | French: 'S3 820 Row 83 Failed To Advance.. Check Qxxx.x French'
  821 = 'S3 821 Row 83 Failed To Return.. Check Qxxx.x Default' | German: 'S3 821 Row 83 Failed To Return.. Check Qxxx.x German' | French: 'S3 821 Row 83 Failed To Return.. Check Qxxx.x French'
  822 = 'S3 822 Row 83 Lost Advance Position... Check Ixxx.x Default' | German: 'S3 822 Row 83 Lost Advance Position... Check Ixxx.x German' | French: 'S3 822 Row 83 Lost Advance Position... Check Ixxx.x French'
  823 = 'S3 823 Row 83 Lost Return Position... Check Ixxx.x Default' | German: 'S3 823 Row 83 Lost Return Position... Check Ixxx.x German' | French: 'S3 823 Row 83 Lost Return Position... Check Ixxx.x French'
  824 = 'S3 824 Row 83 Switch Fault... Check Ixxx.x / Ixxx.x Default' | German: 'S3 824 Row 83 Switch Fault... Check Ixxx.x / Ixxx.x German' | French: 'S3 824 Row 83 Switch Fault... Check Ixxx.x / Ixxx.x French'
  825 = 'S3 825 Row 83 Spare Message Default' | German: 'S3 825 Row 83 Spare Message German' | French: 'S3 825 Row 83 Spare Message French'
  826 = 'S3 826 Row 83 Spare Message Default' | German: 'S3 826 Row 83 Spare Message German' | French: 'S3 826 Row 83 Spare Message French'
  827 = 'S3 827 Row 83 Spare Message Default' | German: 'S3 827 Row 83 Spare Message German' | French: 'S3 827 Row 83 Spare Message French'
  828 = 'S3 828 Row 83 Spare Message Default' | German: 'S3 828 Row 83 Spare Message German' | French: 'S3 828 Row 83 Spare Message French'
  829 = 'S3 829 Row 83 Spare Message Default' | German: 'S3 829 Row 83 Spare Message German' | French: 'S3 829 Row 83 Spare Message French'
  830 = 'S3 830 Row 84 Failed To Advance.. Check Qxxx.x Default' | German: 'S3 830 Row 84 Failed To Advance.. Check Qxxx.x German' | French: 'S3 830 Row 84 Failed To Advance.. Check Qxxx.x French'
  831 = 'S3 831 Row 84 Failed To Return.. Check Qxxx.x Default' | German: 'S3 831 Row 84 Failed To Return.. Check Qxxx.x German' | French: 'S3 831 Row 84 Failed To Return.. Check Qxxx.x French'
  832 = 'S3 832 Row 84 Lost Advance Position... Check Ixxx.x Default' | German: 'S3 832 Row 84 Lost Advance Position... Check Ixxx.x German' | French: 'S3 832 Row 84 Lost Advance Position... Check Ixxx.x French'
  833 = 'S3 833 Row 84 Lost Return Position... Check Ixxx.x Default' | German: 'S3 833 Row 84 Lost Return Position... Check Ixxx.x German' | French: 'S3 833 Row 84 Lost Return Position... Check Ixxx.x French'
  834 = 'S3 834 Row 84 Switch Fault... Check Ixxx.x / Ixxx.x Default' | German: 'S3 834 Row 84 Switch Fault... Check Ixxx.x / Ixxx.x German' | French: 'S3 834 Row 84 Switch Fault... Check Ixxx.x / Ixxx.x French'
  835 = 'S3 835 Row 84 Spare Message Default' | German: 'S3 835 Row 84 Spare Message German' | French: 'S3 835 Row 84 Spare Message French'
  836 = 'S3 836 Row 84 Spare Message Default' | German: 'S3 836 Row 84 Spare Message German' | French: 'S3 836 Row 84 Spare Message French'
  837 = 'S3 837 Row 84 Spare Message Default' | German: 'S3 837 Row 84 Spare Message German' | French: 'S3 837 Row 84 Spare Message French'
  838 = 'S3 838 Row 84 Spare Message Default' | German: 'S3 838 Row 84 Spare Message German' | French: 'S3 838 Row 84 Spare Message French'
  839 = 'S3 839 Row 84 Spare Message Default' | German: 'S3 839 Row 84 Spare Message German' | French: 'S3 839 Row 84 Spare Message French'
  840 = 'S3 840 Row 85 Failed To Advance.. Check Qxxx.x Default' | German: 'S3 840 Row 85 Failed To Advance.. Check Qxxx.x German' | French: 'S3 840 Row 85 Failed To Advance.. Check Qxxx.x French'
  841 = 'S3 841 Row 85 Failed To Return.. Check Qxxx.x Default' | German: 'S3 841 Row 85 Failed To Return.. Check Qxxx.x German' | French: 'S3 841 Row 85 Failed To Return.. Check Qxxx.x French'
  842 = 'S3 842 Row 85 Lost Advance Position... Check Ixxx.x Default' | German: 'S3 842 Row 85 Lost Advance Position... Check Ixxx.x German' | French: 'S3 842 Row 85 Lost Advance Position... Check Ixxx.x French'
  843 = 'S3 843 Row 85 Lost Return Position... Check Ixxx.x Default' | German: 'S3 843 Row 85 Lost Return Position... Check Ixxx.x German' | French: 'S3 843 Row 85 Lost Return Position... Check Ixxx.x French'
  844 = 'S3 844 Row 85 Switch Fault... Check Ixxx.x / Ixxx.x Default' | German: 'S3 844 Row 85 Switch Fault... Check Ixxx.x / Ixxx.x German' | French: 'S3 844 Row 85 Switch Fault... Check Ixxx.x / Ixxx.x French'
  845 = 'S3 845 Row 85 Spare Message Default' | German: 'S3 845 Row 85 Spare Message German' | French: 'S3 845 Row 85 Spare Message French'
  846 = 'S3 846 Row 85 Spare Message Default' | German: 'S3 846 Row 85 Spare Message German' | French: 'S3 846 Row 85 Spare Message French'
  847 = 'S3 847 Row 85 Spare Message Default' | German: 'S3 847 Row 85 Spare Message German' | French: 'S3 847 Row 85 Spare Message French'
  848 = 'S3 848 Row 85 Spare Message Default' | German: 'S3 848 Row 85 Spare Message German' | French: 'S3 848 Row 85 Spare Message French'
  849 = 'S3 849 Row 85 Spare Message Default' | German: 'S3 849 Row 85 Spare Message German' | French: 'S3 849 Row 85 Spare Message French'
  850 = 'S3 850 Row 86 Failed To Advance.. Check Qxxx.x Default' | German: 'S3 850 Row 86 Failed To Advance.. Check Qxxx.x German' | French: 'S3 850 Row 86 Failed To Advance.. Check Qxxx.x French'
  851 = 'S3 851 Row 86 Failed To Return.. Check Qxxx.x Default' | German: 'S3 851 Row 86 Failed To Return.. Check Qxxx.x German' | French: 'S3 851 Row 86 Failed To Return.. Check Qxxx.x French'
  852 = 'S3 852 Row 86 Lost Advance Position... Check Ixxx.x Default' | German: 'S3 852 Row 86 Lost Advance Position... Check Ixxx.x German' | French: 'S3 852 Row 86 Lost Advance Position... Check Ixxx.x French'
  853 = 'S3 853 Row 86 Lost Return Position... Check Ixxx.x Default' | German: 'S3 853 Row 86 Lost Return Position... Check Ixxx.x German' | French: 'S3 853 Row 86 Lost Return Position... Check Ixxx.x French'
  854 = 'S3 854 Row 86 Switch Fault... Check Ixxx.x / Ixxx.x Default' | German: 'S3 854 Row 86 Switch Fault... Check Ixxx.x / Ixxx.x German' | French: 'S3 854 Row 86 Switch Fault... Check Ixxx.x / Ixxx.x French'
  855 = 'S3 855 Row 86 Spare Message Default' | German: 'S3 855 Row 86 Spare Message German' | French: 'S3 855 Row 86 Spare Message French'
  856 = 'S3 856 Row 86 Spare Message Default' | German: 'S3 856 Row 86 Spare Message German' | French: 'S3 856 Row 86 Spare Message French'
  857 = 'S3 857 Row 86 Spare Message Default' | German: 'S3 857 Row 86 Spare Message German' | French: 'S3 857 Row 86 Spare Message French'
  858 = 'S3 858 Row 86 Spare Message Default' | German: 'S3 858 Row 86 Spare Message German' | French: 'S3 858 Row 86 Spare Message French'
  859 = 'S3 859 Row 86 Spare Message Default' | German: 'S3 859 Row 86 Spare Message German' | French: 'S3 859 Row 86 Spare Message French'
  860 = 'S3 860 Row 87 Failed To Advance.. Check Qxxx.x Default' | German: 'S3 860 Row 87 Failed To Advance.. Check Qxxx.x German' | French: 'S3 860 Row 87 Failed To Advance.. Check Qxxx.x French'
  861 = 'S3 861 Row 87 Failed To Return.. Check Qxxx.x Default' | German: 'S3 861 Row 87 Failed To Return.. Check Qxxx.x German' | French: 'S3 861 Row 87 Failed To Return.. Check Qxxx.x French'
  862 = 'S3 862 Row 87 Lost Advance Position... Check Ixxx.x Default' | German: 'S3 862 Row 87 Lost Advance Position... Check Ixxx.x German' | French: 'S3 862 Row 87 Lost Advance Position... Check Ixxx.x French'
  863 = 'S3 863 Row 87 Lost Return Position... Check Ixxx.x Default' | German: 'S3 863 Row 87 Lost Return Position... Check Ixxx.x German' | French: 'S3 863 Row 87 Lost Return Position... Check Ixxx.x French'
  864 = 'S3 864 Row 87 Switch Fault... Check Ixxx.x / Ixxx.x Default' | German: 'S3 864 Row 87 Switch Fault... Check Ixxx.x / Ixxx.x German' | French: 'S3 864 Row 87 Switch Fault... Check Ixxx.x / Ixxx.x French'
  865 = 'S3 865 Row 87 Spare Message Default' | German: 'S3 865 Row 87 Spare Message German' | French: 'S3 865 Row 87 Spare Message French'
  866 = 'S3 866 Row 87 Spare Message Default' | German: 'S3 866 Row 87 Spare Message German' | French: 'S3 866 Row 87 Spare Message French'
  867 = 'S3 867 Row 87 Spare Message Default' | German: 'S3 867 Row 87 Spare Message German' | French: 'S3 867 Row 87 Spare Message French'
  868 = 'S3 868 Row 87 Spare Message Default' | German: 'S3 868 Row 87 Spare Message German' | French: 'S3 868 Row 87 Spare Message French'
  869 = 'S3 869 Row 87 Spare Message Default' | German: 'S3 869 Row 87 Spare Message German' | French: 'S3 869 Row 87 Spare Message French'
  870 = 'S3 870 Row 88 Failed To Advance.. Check Qxxx.x Default' | German: 'S3 870 Row 88 Failed To Advance.. Check Qxxx.x German' | French: 'S3 870 Row 88 Failed To Advance.. Check Qxxx.x French'
  871 = 'S3 871 Row 88 Failed To Return.. Check Qxxx.x Default' | German: 'S3 871 Row 88 Failed To Return.. Check Qxxx.x German' | French: 'S3 871 Row 88 Failed To Return.. Check Qxxx.x French'
  872 = 'S3 872 Row 88 Lost Advance Position... Check Ixxx.x Default' | German: 'S3 872 Row 88 Lost Advance Position... Check Ixxx.x German' | French: 'S3 872 Row 88 Lost Advance Position... Check Ixxx.x French'
  873 = 'S3 873 Row 88 Lost Return Position... Check Ixxx.x Default' | German: 'S3 873 Row 88 Lost Return Position... Check Ixxx.x German' | French: 'S3 873 Row 88 Lost Return Position... Check Ixxx.x French'
  874 = 'S3 874 Row 88 Switch Fault... Check Ixxx.x / Ixxx.x Default' | German: 'S3 874 Row 88 Switch Fault... Check Ixxx.x / Ixxx.x German' | French: 'S3 874 Row 88 Switch Fault... Check Ixxx.x / Ixxx.x French'
  875 = 'S3 875 Row 88 Spare Message Default' | German: 'S3 875 Row 88 Spare Message German' | French: 'S3 875 Row 88 Spare Message French'
  876 = 'S3 876 Row 88 Spare Message Default' | German: 'S3 876 Row 88 Spare Message German' | French: 'S3 876 Row 88 Spare Message French'
  877 = 'S3 877 Row 88 Spare Message Default' | German: 'S3 877 Row 88 Spare Message German' | French: 'S3 877 Row 88 Spare Message French'
  878 = 'S3 878 Row 88 Spare Message Default' | German: 'S3 878 Row 88 Spare Message German' | French: 'S3 878 Row 88 Spare Message French'
  879 = 'S3 879 Row 88 Spare Message Default' | German: 'S3 879 Row 88 Spare Message German' | French: 'S3 879 Row 88 Spare Message French'
  880 = 'S3 880 Row 89 Failed To Advance.. Check Qxxx.x Default' | German: 'S3 880 Row 89 Failed To Advance.. Check Qxxx.x German' | French: 'S3 880 Row 89 Failed To Advance.. Check Qxxx.x French'
  881 = 'S3 881 Row 89 Failed To Return.. Check Qxxx.x Default' | German: 'S3 881 Row 89 Failed To Return.. Check Qxxx.x German' | French: 'S3 881 Row 89 Failed To Return.. Check Qxxx.x French'
  882 = 'S3 882 Row 89 Lost Advance Position... Check Ixxx.x Default' | German: 'S3 882 Row 89 Lost Advance Position... Check Ixxx.x German' | French: 'S3 882 Row 89 Lost Advance Position... Check Ixxx.x French'
  883 = 'S3 883 Row 89 Lost Return Position... Check Ixxx.x Default' | German: 'S3 883 Row 89 Lost Return Position... Check Ixxx.x German' | French: 'S3 883 Row 89 Lost Return Position... Check Ixxx.x French'
  884 = 'S3 884 Row 89 Switch Fault... Check Ixxx.x / Ixxx.x Default' | German: 'S3 884 Row 89 Switch Fault... Check Ixxx.x / Ixxx.x German' | French: 'S3 884 Row 89 Switch Fault... Check Ixxx.x / Ixxx.x French'
  885 = 'S3 885 Row 89 Spare Message Default' | German: 'S3 885 Row 89 Spare Message German' | French: 'S3 885 Row 89 Spare Message French'
  886 = 'S3 886 Row 89 Spare Message Default' | German: 'S3 886 Row 89 Spare Message German' | French: 'S3 886 Row 89 Spare Message French'
  887 = 'S3 887 Row 89 Spare Message Default' | German: 'S3 887 Row 89 Spare Message German' | French: 'S3 887 Row 89 Spare Message French'
  888 = 'S3 888 Row 89 Spare Message Default' | German: 'S3 888 Row 89 Spare Message German' | French: 'S3 888 Row 89 Spare Message French'
  889 = 'S3 889 Row 89 Spare Message Default' | German: 'S3 889 Row 89 Spare Message German' | French: 'S3 889 Row 89 Spare Message French'
  890 = 'S3 890 Row 90 Failed To Advance.. Check Qxxx.x Default' | German: 'S3 890 Row 90 Failed To Advance.. Check Qxxx.x German' | French: 'S3 890 Row 90 Failed To Advance.. Check Qxxx.x French'
  891 = 'S3 891 Row 90 Failed To Return.. Check Qxxx.x Default' | German: 'S3 891 Row 90 Failed To Return.. Check Qxxx.x German' | French: 'S3 891 Row 90 Failed To Return.. Check Qxxx.x French'
  892 = 'S3 892 Row 90 Lost Advance Position... Check Ixxx.x Default' | German: 'S3 892 Row 90 Lost Advance Position... Check Ixxx.x German' | French: 'S3 892 Row 90 Lost Advance Position... Check Ixxx.x French'
  893 = 'S3 893 Row 90 Lost Return Position... Check Ixxx.x Default' | German: 'S3 893 Row 90 Lost Return Position... Check Ixxx.x German' | French: 'S3 893 Row 90 Lost Return Position... Check Ixxx.x French'
  894 = 'S3 894 Row 90 Switch Fault... Check Ixxx.x / Ixxx.x Default' | German: 'S3 894 Row 90 Switch Fault... Check Ixxx.x / Ixxx.x German' | French: 'S3 894 Row 90 Switch Fault... Check Ixxx.x / Ixxx.x French'
  895 = 'S3 895 Row 90 Spare Message Default' | German: 'S3 895 Row 90 Spare Message German' | French: 'S3 895 Row 90 Spare Message French'
  896 = 'S3 896 Row 90 Spare Message Default' | German: 'S3 896 Row 90 Spare Message German' | French: 'S3 896 Row 90 Spare Message French'
  897 = 'S3 897 Row 90 Spare Message Default' | German: 'S3 897 Row 90 Spare Message German' | French: 'S3 897 Row 90 Spare Message French'
  898 = 'S3 898 Row 90 Spare Message Default' | German: 'S3 898 Row 90 Spare Message German' | French: 'S3 898 Row 90 Spare Message French'
  899 = 'S3 899 Row 90 Spare Message Default' | German: 'S3 899 Row 90 Spare Message German' | French: 'S3 899 Row 90 Spare Message French'
  900 = 'S3 900 Row 91 Failed To Advance.. Check Qxxx.x Default' | German: 'S3 900 Row 91 Failed To Advance.. Check Qxxx.x German' | French: 'S3 900 Row 91 Failed To Advance.. Check Qxxx.x French'
  901 = 'S3 901 Row 91 Failed To Return.. Check Qxxx.x Default' | German: 'S3 901 Row 91 Failed To Return.. Check Qxxx.x German' | French: 'S3 901 Row 91 Failed To Return.. Check Qxxx.x French'
  902 = 'S3 902 Row 91 Lost Advance Position... Check Ixxx.x Default' | German: 'S3 902 Row 91 Lost Advance Position... Check Ixxx.x German' | French: 'S3 902 Row 91 Lost Advance Position... Check Ixxx.x French'
  903 = 'S3 903 Row 91 Lost Return Position... Check Ixxx.x Default' | German: 'S3 903 Row 91 Lost Return Position... Check Ixxx.x German' | French: 'S3 903 Row 91 Lost Return Position... Check Ixxx.x French'
  904 = 'S3 904 Row 91 Switch Fault... Check Ixxx.x / Ixxx.x Default' | German: 'S3 904 Row 91 Switch Fault... Check Ixxx.x / Ixxx.x German' | French: 'S3 904 Row 91 Switch Fault... Check Ixxx.x / Ixxx.x French'
  905 = 'S3 905 Row 91 Spare Message Default' | German: 'S3 905 Row 91 Spare Message German' | French: 'S3 905 Row 91 Spare Message French'
  906 = 'S3 906 Row 91 Spare Message Default' | German: 'S3 906 Row 91 Spare Message German' | French: 'S3 906 Row 91 Spare Message French'
  907 = 'S3 907 Row 91 Spare Message Default' | German: 'S3 907 Row 91 Spare Message German' | French: 'S3 907 Row 91 Spare Message French'
  908 = 'S3 908 Row 91 Spare Message Default' | German: 'S3 908 Row 91 Spare Message German' | French: 'S3 908 Row 91 Spare Message French'
  909 = 'S3 909 Row 91 Spare Message Default' | German: 'S3 909 Row 91 Spare Message German' | French: 'S3 909 Row 91 Spare Message French'
  910 = 'S3 910 Row 92 Failed To Advance.. Check Qxxx.x Default' | German: 'S3 910 Row 92 Failed To Advance.. Check Qxxx.x German' | French: 'S3 910 Row 92 Failed To Advance.. Check Qxxx.x French'
  911 = 'S3 911 Row 92 Failed To Return.. Check Qxxx.x Default' | German: 'S3 911 Row 92 Failed To Return.. Check Qxxx.x German' | French: 'S3 911 Row 92 Failed To Return.. Check Qxxx.x French'
  912 = 'S3 912 Row 92 Lost Advance Position... Check Ixxx.x Default' | German: 'S3 912 Row 92 Lost Advance Position... Check Ixxx.x German' | French: 'S3 912 Row 92 Lost Advance Position... Check Ixxx.x French'
  913 = 'S3 913 Row 92 Lost Return Position... Check Ixxx.x Default' | German: 'S3 913 Row 92 Lost Return Position... Check Ixxx.x German' | French: 'S3 913 Row 92 Lost Return Position... Check Ixxx.x French'
  914 = 'S3 914 Row 92 Switch Fault... Check Ixxx.x / Ixxx.x Default' | German: 'S3 914 Row 92 Switch Fault... Check Ixxx.x / Ixxx.x German' | French: 'S3 914 Row 92 Switch Fault... Check Ixxx.x / Ixxx.x French'
  915 = 'S3 915 Row 92 Spare Message Default' | German: 'S3 915 Row 92 Spare Message German' | French: 'S3 915 Row 92 Spare Message French'
  916 = 'S3 916 Row 92 Spare Message Default' | German: 'S3 916 Row 92 Spare Message German' | French: 'S3 916 Row 92 Spare Message French'
  917 = 'S3 917 Row 92 Spare Message Default' | German: 'S3 917 Row 92 Spare Message German' | French: 'S3 917 Row 92 Spare Message French'
  918 = 'S3 918 Row 92 Spare Message Default' | German: 'S3 918 Row 92 Spare Message German' | French: 'S3 918 Row 92 Spare Message French'
  919 = 'S3 919 Row 92 Spare Message Default' | German: 'S3 919 Row 92 Spare Message German' | French: 'S3 919 Row 92 Spare Message French'
  920 = 'S3 920 Row 93 Failed To Advance.. Check Qxxx.x Default' | German: 'S3 920 Row 93 Failed To Advance.. Check Qxxx.x German' | French: 'S3 920 Row 93 Failed To Advance.. Check Qxxx.x French'
  921 = 'S3 921 Row 93 Failed To Return.. Check Qxxx.x Default' | German: 'S3 921 Row 93 Failed To Return.. Check Qxxx.x German' | French: 'S3 921 Row 93 Failed To Return.. Check Qxxx.x French'
  922 = 'S3 922 Row 93 Lost Advance Position... Check Ixxx.x Default' | German: 'S3 922 Row 93 Lost Advance Position... Check Ixxx.x German' | French: 'S3 922 Row 93 Lost Advance Position... Check Ixxx.x French'
  923 = 'S3 923 Row 93 Lost Return Position... Check Ixxx.x Default' | German: 'S3 923 Row 93 Lost Return Position... Check Ixxx.x German' | French: 'S3 923 Row 93 Lost Return Position... Check Ixxx.x French'
  924 = 'S3 924 Row 93 Switch Fault... Check Ixxx.x / Ixxx.x Default' | German: 'S3 924 Row 93 Switch Fault... Check Ixxx.x / Ixxx.x German' | French: 'S3 924 Row 93 Switch Fault... Check Ixxx.x / Ixxx.x French'
  925 = 'S3 925 Row 93 Spare Message Default' | German: 'S3 925 Row 93 Spare Message German' | French: 'S3 925 Row 93 Spare Message French'
  926 = 'S3 926 Row 93 Spare Message Default' | German: 'S3 926 Row 93 Spare Message German' | French: 'S3 926 Row 93 Spare Message French'
  927 = 'S3 927 Row 93 Spare Message Default' | German: 'S3 927 Row 93 Spare Message German' | French: 'S3 927 Row 93 Spare Message French'
  928 = 'S3 928 Row 93 Spare Message Default' | German: 'S3 928 Row 93 Spare Message German' | French: 'S3 928 Row 93 Spare Message French'
  929 = 'S3 929 Row 93 Spare Message Default' | German: 'S3 929 Row 93 Spare Message German' | French: 'S3 929 Row 93 Spare Message French'
  930 = 'S3 930 Row 94 Failed To Advance.. Check Qxxx.x Default' | German: 'S3 930 Row 94 Failed To Advance.. Check Qxxx.x German' | French: 'S3 930 Row 94 Failed To Advance.. Check Qxxx.x French'
  931 = 'S3 931 Row 94 Failed To Return.. Check Qxxx.x Default' | German: 'S3 931 Row 94 Failed To Return.. Check Qxxx.x German' | French: 'S3 931 Row 94 Failed To Return.. Check Qxxx.x French'
  932 = 'S3 932 Row 94 Lost Advance Position... Check Ixxx.x Default' | German: 'S3 932 Row 94 Lost Advance Position... Check Ixxx.x German' | French: 'S3 932 Row 94 Lost Advance Position... Check Ixxx.x French'
  933 = 'S3 933 Row 94 Lost Return Position... Check Ixxx.x Default' | German: 'S3 933 Row 94 Lost Return Position... Check Ixxx.x German' | French: 'S3 933 Row 94 Lost Return Position... Check Ixxx.x French'
  934 = 'S3 934 Row 94 Switch Fault... Check Ixxx.x / Ixxx.x Default' | German: 'S3 934 Row 94 Switch Fault... Check Ixxx.x / Ixxx.x German' | French: 'S3 934 Row 94 Switch Fault... Check Ixxx.x / Ixxx.x French'
  935 = 'S3 935 Row 94 Spare Message Default' | German: 'S3 935 Row 94 Spare Message German' | French: 'S3 935 Row 94 Spare Message French'
  936 = 'S3 936 Row 94 Spare Message Default' | German: 'S3 936 Row 94 Spare Message German' | French: 'S3 936 Row 94 Spare Message French'
  937 = 'S3 937 Row 94 Spare Message Default' | German: 'S3 937 Row 94 Spare Message German' | French: 'S3 937 Row 94 Spare Message French'
  938 = 'S3 938 Row 94 Spare Message Default' | German: 'S3 938 Row 94 Spare Message German' | French: 'S3 938 Row 94 Spare Message French'
  939 = 'S3 939 Row 94 Spare Message Default' | German: 'S3 939 Row 94 Spare Message German' | French: 'S3 939 Row 94 Spare Message French'
  940 = 'S3 940 Row 95 Failed To Advance.. Check Qxxx.x Default' | German: 'S3 940 Row 95 Failed To Advance.. Check Qxxx.x German' | French: 'S3 940 Row 95 Failed To Advance.. Check Qxxx.x French'
  941 = 'S3 941 Row 95 Failed To Return.. Check Qxxx.x Default' | German: 'S3 941 Row 95 Failed To Return.. Check Qxxx.x German' | French: 'S3 941 Row 95 Failed To Return.. Check Qxxx.x French'
  942 = 'S3 942 Row 95 Lost Advance Position... Check Ixxx.x Default' | German: 'S3 942 Row 95 Lost Advance Position... Check Ixxx.x German' | French: 'S3 942 Row 95 Lost Advance Position... Check Ixxx.x French'
  943 = 'S3 943 Row 95 Lost Return Position... Check Ixxx.x Default' | German: 'S3 943 Row 95 Lost Return Position... Check Ixxx.x German' | French: 'S3 943 Row 95 Lost Return Position... Check Ixxx.x French'
  944 = 'S3 944 Row 95 Switch Fault... Check Ixxx.x / Ixxx.x Default' | German: 'S3 944 Row 95 Switch Fault... Check Ixxx.x / Ixxx.x German' | French: 'S3 944 Row 95 Switch Fault... Check Ixxx.x / Ixxx.x French'
  945 = 'S3 945 Row 95 Spare Message Default' | German: 'S3 945 Row 95 Spare Message German' | French: 'S3 945 Row 95 Spare Message French'
  946 = 'S3 946 Row 95 Spare Message Default' | German: 'S3 946 Row 95 Spare Message German' | French: 'S3 946 Row 95 Spare Message French'
  947 = 'S3 947 Row 95 Spare Message Default' | German: 'S3 947 Row 95 Spare Message German' | French: 'S3 947 Row 95 Spare Message French'
  948 = 'S3 948 Row 95 Spare Message Default' | German: 'S3 948 Row 95 Spare Message German' | French: 'S3 948 Row 95 Spare Message French'
  949 = 'S3 949 Row 95 Spare Message Default' | German: 'S3 949 Row 95 Spare Message German' | French: 'S3 949 Row 95 Spare Message French'
  950 = 'S3 950 Row 96 Failed To Advance.. Check Qxxx.x Default' | German: 'S3 950 Row 96 Failed To Advance.. Check Qxxx.x German' | French: 'S3 950 Row 96 Failed To Advance.. Check Qxxx.x French'
  951 = 'S3 951 Row 96 Failed To Return.. Check Qxxx.x Default' | German: 'S3 951 Row 96 Failed To Return.. Check Qxxx.x German' | French: 'S3 951 Row 96 Failed To Return.. Check Qxxx.x French'
  952 = 'S3 952 Row 96 Lost Advance Position... Check Ixxx.x Default' | German: 'S3 952 Row 96 Lost Advance Position... Check Ixxx.x German' | French: 'S3 952 Row 96 Lost Advance Position... Check Ixxx.x French'
  953 = 'S3 953 Row 96 Lost Return Position... Check Ixxx.x Default' | German: 'S3 953 Row 96 Lost Return Position... Check Ixxx.x German' | French: 'S3 953 Row 96 Lost Return Position... Check Ixxx.x French'
  954 = 'S3 954 Row 96 Switch Fault... Check Ixxx.x / Ixxx.x Default' | German: 'S3 954 Row 96 Switch Fault... Check Ixxx.x / Ixxx.x German' | French: 'S3 954 Row 96 Switch Fault... Check Ixxx.x / Ixxx.x French'
  955 = 'S3 955 Row 96 Spare Message Default' | German: 'S3 955 Row 96 Spare Message German' | French: 'S3 955 Row 96 Spare Message French'
  956 = 'S3 956 Row 96 Spare Message Default' | German: 'S3 956 Row 96 Spare Message German' | French: 'S3 956 Row 96 Spare Message French'
  957 = 'S3 957 Row 96 Spare Message Default' | German: 'S3 957 Row 96 Spare Message German' | French: 'S3 957 Row 96 Spare Message French'
  958 = 'S3 958 Row 96 Spare Message Default' | German: 'S3 958 Row 96 Spare Message German' | French: 'S3 958 Row 96 Spare Message French'
  959 = 'S3 959 Row 96 Spare Message Default' | German: 'S3 959 Row 96 Spare Message German' | French: 'S3 959 Row 96 Spare Message French'
  960 = 'S3 960 Row 97 Failed To Advance.. Check Qxxx.x Default' | German: 'S3 960 Row 97 Failed To Advance.. Check Qxxx.x German' | French: 'S3 960 Row 97 Failed To Advance.. Check Qxxx.x French'
  961 = 'S3 961 Row 97 Failed To Return.. Check Qxxx.x Default' | German: 'S3 961 Row 97 Failed To Return.. Check Qxxx.x German' | French: 'S3 961 Row 97 Failed To Return.. Check Qxxx.x French'
  962 = 'S3 962 Row 97 Lost Advance Position... Check Ixxx.x Default' | German: 'S3 962 Row 97 Lost Advance Position... Check Ixxx.x German' | French: 'S3 962 Row 97 Lost Advance Position... Check Ixxx.x French'
  963 = 'S3 963 Row 97 Lost Return Position... Check Ixxx.x Default' | German: 'S3 963 Row 97 Lost Return Position... Check Ixxx.x German' | French: 'S3 963 Row 97 Lost Return Position... Check Ixxx.x French'
  964 = 'S3 964 Row 97 Switch Fault... Check Ixxx.x / Ixxx.x Default' | German: 'S3 964 Row 97 Switch Fault... Check Ixxx.x / Ixxx.x German' | French: 'S3 964 Row 97 Switch Fault... Check Ixxx.x / Ixxx.x French'
  965 = 'S3 965 Row 97 Spare Message Default' | German: 'S3 965 Row 97 Spare Message German' | French: 'S3 965 Row 97 Spare Message French'
  966 = 'S3 966 Row 97 Spare Message Default' | German: 'S3 966 Row 97 Spare Message German' | French: 'S3 966 Row 97 Spare Message French'
  967 = 'S3 967 Row 97 Spare Message Default' | German: 'S3 967 Row 97 Spare Message German' | French: 'S3 967 Row 97 Spare Message French'
  968 = 'S3 968 Row 97 Spare Message Default' | German: 'S3 968 Row 97 Spare Message German' | French: 'S3 968 Row 97 Spare Message French'
  969 = 'S3 969 Row 97 Spare Message Default' | German: 'S3 969 Row 97 Spare Message German' | French: 'S3 969 Row 97 Spare Message French'
  970 = 'S3 970 Row 98 Failed To Advance.. Check Qxxx.x Default' | German: 'S3 970 Row 98 Failed To Advance.. Check Qxxx.x German' | French: 'S3 970 Row 98 Failed To Advance.. Check Qxxx.x French'
  971 = 'S3 971 Row 98 Failed To Return.. Check Qxxx.x Default' | German: 'S3 971 Row 98 Failed To Return.. Check Qxxx.x German' | French: 'S3 971 Row 98 Failed To Return.. Check Qxxx.x French'
  972 = 'S3 972 Row 98 Lost Advance Position... Check Ixxx.x Default' | German: 'S3 972 Row 98 Lost Advance Position... Check Ixxx.x German' | French: 'S3 972 Row 98 Lost Advance Position... Check Ixxx.x French'
  973 = 'S3 973 Row 98 Lost Return Position... Check Ixxx.x Default' | German: 'S3 973 Row 98 Lost Return Position... Check Ixxx.x German' | French: 'S3 973 Row 98 Lost Return Position... Check Ixxx.x French'
  974 = 'S3 974 Row 98 Switch Fault... Check Ixxx.x / Ixxx.x Default' | German: 'S3 974 Row 98 Switch Fault... Check Ixxx.x / Ixxx.x German' | French: 'S3 974 Row 98 Switch Fault... Check Ixxx.x / Ixxx.x French'
  975 = 'S3 975 Row 98 Spare Message Default' | German: 'S3 975 Row 98 Spare Message German' | French: 'S3 975 Row 98 Spare Message French'
  976 = 'S3 976 Row 98 Spare Message Default' | German: 'S3 976 Row 98 Spare Message German' | French: 'S3 976 Row 98 Spare Message French'
  977 = 'S3 977 Row 98 Spare Message Default' | German: 'S3 977 Row 98 Spare Message German' | French: 'S3 977 Row 98 Spare Message French'
  978 = 'S3 978 Row 98 Spare Message Default' | German: 'S3 978 Row 98 Spare Message German' | French: 'S3 978 Row 98 Spare Message French'
  979 = 'S3 979 Row 98 Spare Message Default' | German: 'S3 979 Row 98 Spare Message German' | French: 'S3 979 Row 98 Spare Message French'
  980 = 'S3 980 Row 99 Failed To Advance.. Check Qxxx.x Default' | German: 'S3 980 Row 99 Failed To Advance.. Check Qxxx.x German' | French: 'S3 980 Row 99 Failed To Advance.. Check Qxxx.x French'
  981 = 'S3 981 Row 99 Failed To Return.. Check Qxxx.x Default' | German: 'S3 981 Row 99 Failed To Return.. Check Qxxx.x German' | French: 'S3 981 Row 99 Failed To Return.. Check Qxxx.x French'
  982 = 'S3 982 Row 99 Lost Advance Position... Check Ixxx.x Default' | German: 'S3 982 Row 99 Lost Advance Position... Check Ixxx.x German' | French: 'S3 982 Row 99 Lost Advance Position... Check Ixxx.x French'
  983 = 'S3 983 Row 99 Lost Return Position... Check Ixxx.x Default' | German: 'S3 983 Row 99 Lost Return Position... Check Ixxx.x German' | French: 'S3 983 Row 99 Lost Return Position... Check Ixxx.x French'
  984 = 'S3 984 Row 99 Switch Fault... Check Ixxx.x / Ixxx.x Default' | German: 'S3 984 Row 99 Switch Fault... Check Ixxx.x / Ixxx.x German' | French: 'S3 984 Row 99 Switch Fault... Check Ixxx.x / Ixxx.x French'
  985 = 'S3 985 Row 99 Spare Message Default' | German: 'S3 985 Row 99 Spare Message German' | French: 'S3 985 Row 99 Spare Message French'
  986 = 'S3 986 Row 99 Spare Message Default' | German: 'S3 986 Row 99 Spare Message German' | French: 'S3 986 Row 99 Spare Message French'
  987 = 'S3 987 Row 99 Spare Message Default' | German: 'S3 987 Row 99 Spare Message German' | French: 'S3 987 Row 99 Spare Message French'
  988 = 'S3 988 Row 99 Spare Message Default' | German: 'S3 988 Row 99 Spare Message German' | French: 'S3 988 Row 99 Spare Message French'
  989 = 'S3 989 Row 99 Spare Message Default' | German: 'S3 989 Row 99 Spare Message German' | French: 'S3 989 Row 99 Spare Message French'
  990 = 'S3 990 Row 100 Failed To Advance.. Check Qxxx.x Default' | German: 'S3 990 Row 100 Failed To Advance.. Check Qxxx.x German' | French: 'S3 990 Row 100 Failed To Advance.. Check Qxxx.x French'
  991 = 'S3 991 Row 100 Failed To Return.. Check Qxxx.x Default' | German: 'S3 991 Row 100 Failed To Return.. Check Qxxx.x German' | French: 'S3 991 Row 100 Failed To Return.. Check Qxxx.x French'
  992 = 'S3 992 Row 100 Lost Advance Position... Check Ixxx.x Default' | German: 'S3 992 Row 100 Lost Advance Position... Check Ixxx.x German' | French: 'S3 992 Row 100 Lost Advance Position... Check Ixxx.x French'
  993 = 'S3 993 Row 100 Lost Return Position... Check Ixxx.x Default' | German: 'S3 993 Row 100 Lost Return Position... Check Ixxx.x German' | French: 'S3 993 Row 100 Lost Return Position... Check Ixxx.x French'
  994 = 'S3 994 Row 100 Switch Fault... Check Ixxx.x / Ixxx.x Default' | German: 'S3 994 Row 100 Switch Fault... Check Ixxx.x / Ixxx.x German' | French: 'S3 994 Row 100 Switch Fault... Check Ixxx.x / Ixxx.x French'
  995 = 'S3 995 Row 100 Spare Message Default' | German: 'S3 995 Row 100 Spare Message German' | French: 'S3 995 Row 100 Spare Message French'
  996 = 'S3 996 Row 100 Spare Message Default' | German: 'S3 996 Row 100 Spare Message German' | French: 'S3 996 Row 100 Spare Message French'
  997 = 'S3 997 Row 100 Spare Message Default' | German: 'S3 997 Row 100 Spare Message German' | French: 'S3 997 Row 100 Spare Message French'
  998 = 'S3 998 Row 100 Spare Message Default' | German: 'S3 998 Row 100 Spare Message German' | French: 'S3 998 Row 100 Spare Message French'
  999 = 'S3 999 Row 100 Spare Message Default' | German: 'S3 999 Row 100 Spare Message German' | French: 'S3 999 Row 100 Spare Message French'
  1000 = 'S3_Alarms Default 1000' | German: 'S3_Alarms German 1000' | French: 'S3_Alarms French 1000'
   = ''
END_TEXTLIST

(* stored: Version 1.1.0.1, ProductVersion 3.1.4024.12
   TextList S3_Alarms: Id {f3fe854b-464f-4295-8a79-c774d357aaac} *)
